Fanuc TP program (LS listing): KFLINE.LS

/PROG  KFLINE
/ATTR
OWNER		= MNEDITOR;
COMMENT		= "KfLine";
PROG_SIZE	= 0;
CREATE		= DATE 26-01-01  TIME 00:00:00;
MODIFIED	= DATE 26-01-01  TIME 00:00:00;
FILE_NAME	= ;
VERSION		= 0;
LINE_COUNT	= 2;
MEMORY_SIZE	= 0;
PROTECT		= READ_WRITE;
TCD:  STACK_SIZE	= 0,
      TASK_PRIORITY	= 50,
      TIME_SLICE	= 0,
      BUSY_LAMP_OFF	= 0,
      ABORT_REQUEST	= 0,
      PAUSE_REQUEST	= 0;
DEFAULT_GROUP	= 1,*,*,*,*;
CONTROL_CODE	= 00000000 00000000;
/MN
   1:  !RAPID KarelFileProbe.KfLine ;
   2:  CALL CA_FILE(2,2,1,'[',AR[1],'] ',AR[2]) ;
/POS
/END
